PROGRAM MAIN
VAR

END_VAR



PRG_1();

END_PROGRAM

(* stored: Version 1.1.0.1, ProductVersion 3.1.4024.4
   POU MAIN: Id {abdead8a-7cdd-4344-829d-9a9b4244d437}, SpecialFunc None *)
